// TIA Portal project "SimuladorPart2" (V15)

(* hardware
DEVICE "S7-1200 station_1"  S7-1200 Station
   slot 0: "Rack_0"  S7-1200 Rack  Rack  V1.0
   slot 1: "PLC_1"  CPU 1214C DC/DC/DC  6ES7 214-1AG40-0XB0  V4.2
   slot 2: "DI 8x24VDC_1"  SM 1221 DI8 x 24VDC  6ES7 221-1BF30-0XB0  V1.0
*)

// ===== PLC "PLC_1"  CPU 1214C DC/DC/DC =====

VAR_GLOBAL   // PLC tag table "Default tag table"
   ""BtnStop"" AT %I0.0 : Bool;
   ""BtnStart"" AT %I0.1 : Bool;
   ""S2Capacitivo"" AT %I0.2 : Bool;
   ""S1Indutivo"" AT %I0.3 : Bool;
   ""S3Pequeno"" AT %I0.4 : Bool;
   ""S4Medio"" AT %I0.5 : Bool;
   ""S5Grande"" AT %I0.6 : Bool;
   ""Resetar defeito"" AT %I0.7 : Bool;
   ""S6_FimDeCurso"" AT %I1.0 : Bool;
   ""Reed_Switch1"" AT %I1.1 : Bool;
   ""Reed_Switch2"" AT %I1.2 : Bool;
   ""Reed_Switch3"" AT %I1.3 : Bool;
   ""SnOtico_Grande"" AT %I1.4 : Bool;
   ""SnOtico_Medio"" AT %I1.5 : Bool;
   ""SnOtico_Pequeno"" AT %I8.0 : Bool;
   ""Motor1"" AT %Q0.1 : Bool;
   ""LampadaDefeito"" AT %Q0.2 : Bool;
   ""Soleoneide1"" AT %Q0.3 : Bool;
   ""Soleoneide2"" AT %Q0.4 : Bool;
   ""Soleoneide3"" AT %Q0.5 : Bool;
END_VAR